Fanuc KAREL source: kt00943.KL

PROGRAM KT00943
%STACKSIZE=65535
%PRIORITY=65535
%NOLOCKGROUP
VAR
ENTRY : INTEGER
PNAME : STRING[80]
VNAME : STRING[80]
STATUS : INTEGER
-- UNRESOLVED DECLARATIONS (source type spelling not recovered)
-- VALUE : TYPE_0x0013 (type_u16=0x0013)
BEGIN
ENTRY=0
PNAME=''
VNAME='VALUE'
GET_VAR(ENTRY,PNAME,VNAME,VALUE,STATUS)
END KT00943
